{attribute 'linkalways'} 
{attribute 'no_explicit_call' := 'This FB is a CLASS and must be accessed using methods or properties'}
{attribute 'enable_dynamic_creation'}
FUNCTION_BLOCK ABSTRACT MiddlewareBase implements I_Middleware
VAR
	_next : I_Middleware;
END_VAR

METHOD PUBLIC ABSTRACT Handle
VAR_INPUT
	Request : I_Request;
	Response : I_ServerResponse;
END_VAR
// Call next to pass the request and response to the next handler
// Next(Request, Response);
END_METHOD

METHOD PROTECTED Next
VAR_INPUT
	Request : I_Request;
	Response : I_ServerResponse;
END_VAR
IF _next = 0 THEN
	RETURN;
END_IF

_next.Handle(Request, Response);
END_METHOD

PROPERTY PUBLIC NextMiddleware : I_Middleware
GET
NextMiddleware := _next;
END_GET
SET
_next := NextMiddleware;
END_SET
END_PROPERTY

END_FUNCTION_BLOCK

(* stored: Version 1.1.0.1, ProductVersion 3.1.4024.12
   POU MiddlewareBase: Id {af066795-5139-47ab-af4d-eab87d77ce03}, SpecialFunc None
   Folder Protected: Id {8176d192-b96d-4c65-b3f4-90e3ed32eac3}
   Method Handle: Id {069e2687-0b1c-48a5-ae7d-c4f3322e6443}
   Method Next: Id {c88c5869-feda-47f4-9f7a-877e6399c98f}
   Property NextMiddleware: Id {ccb192db-e3b8-4503-8eb3-1e0abedb5db0}
   Get Get: Id {4d98b946-e60e-4f0d-a625-243010104109}
   Set Set: Id {623f2f3f-2b07-459b-b91e-a072961318ea} *)
